DATA_BLOCK "ST10_Flow6_FixtureCodeScan_iDB"
{ S7_Optimized_Access := 'TRUE' }
VERSION : 0.1
NON_RETAIN
"ST10_Flow6_ToolCodeScan"

BEGIN

END_DATA_BLOCK

